{attribute 'strict'}
{attribute 'to_string'}
TYPE E_MessageType :
(
  eMessageEmpty,
  eMessageError,
  eMessageWarning,
  eMessageInfo,
  eMessageVerbose
)DINT;
END_TYPE

(* stored: Version 1.1.0.1
   DUT E_MessageType: Id {e08552b9-5432-4d71-a241-cf7e1f8fb21c} *)
